// TIA Portal V17 export
// export: Created 2023-05-07T12:12:23.5223812Z, ExportSetting WithDefaults, DisplayName Totally Integrated Automation Portal, DisplayVersion V17, DisplayName TIA Portal Openness, DisplayVersion V17, DisplayName TIA Portal Version Control Interface, DisplayVersion V17, DisplayName TIA Portal Test Suite Advanced, DisplayVersion V17, DisplayName STEP 7 Professional, DisplayVersion V17, DisplayName SIMATIC Energy Suite, DisplayVersion V17, DisplayName STEP 7 Safety, DisplayVersion V17, DisplayName WinCC Professional, DisplayVersion V17
DATA_BLOCK "Object_DB"   // DB13
VERSION : 0.1
// stored: AutoNumber true, InstanceOfName Object, InstanceOfType FB
"Object"
   // VAR_INPUT
   //    r : Real;
   //    disruption : Real;
   // END_VAR
   // VAR_OUTPUT
   //    y : Real;
   // END_VAR
   // VAR
   //    x_array : Array[0..2] of Real;
   //    y_array : Array[0..2] of Real;
   // END_VAR
BEGIN
END_DATA_BLOCK
